PROGRAM MAIN
VAR
	fbMachine : FB_Machine;	

	Dummy : BOOL := FALSE;
	bTest: BOOL := FALSE;
END_VAR

// =========================================================

fbMachine();

// =========================================================



//GVL_SA.Motor1.UpdateAll();
GVL_SA.Motor1();

GVL_SA.Motor1.bStateEnable := TRUE;

{IF defined (Pyrometer_Motor)}
	bTest := TRUE;
{END_IF}

Dummy	:= TRUE;

END_PROGRAM

(* stored: Version 1.1.0.1, ProductVersion 3.1.4024.11
   POU MAIN: Id {1c4fe094-ad65-4615-9ae0-9ca5c10a1bc8}, SpecialFunc None *)
